(* Logix 5000 project; controller Transcat_L33ER vendor 1 type 14 code 107 rev 32.11; software revision 32.02; part 4 of 5 *)
(* tags used below, declared in another part *)
   alwaysOFF : BOOL;
   AnyAutoDeviceInterlock : BOOL;   // Any device in Auto interlocked
   AnyAutoRun : BOOL;   // Bit that in on if ANY device is placed into Auto run (to signal pre-start beed)
   AnyDeviceInterlock : BOOL;   // Any device is interlocked
   AnyManualRun : BOOL;   // Bit that in on if ANY device is placed into manual run (to signal pre-start beed)
   Auto_Run_All_Interlock : BOOL;   // Bit to interlock all devices running in Auto
   BeaconBlueLight : ALIAS FOR TC_Remote_IO:3:O.3;   // Blue Beacon Light
   BeaconGreenLight : ALIAS FOR TC_Remote_IO:3:O.2;   // Green Beacon Light
   BeaconRedLight : ALIAS FOR TC_Remote_IO:3:O.0;   // Red Beacon Light
   BeaconYellowLight : ALIAS FOR TC_Remote_IO:3:O.1;   // Yellow Beacon Light
   Beep : BOOL;   // Bit to Activte Beacon Alarm
   BeepNew : ALIAS FOR TC_Remote_IO:3:O.4;
   Device : Device[20];
   EstopActive : BOOL;   // E
   EstopFalutResetTOF : TIMER;   // Timer to hold reset bit to allow all drives to reset
   EStopReset_OS : BOOL;   // Storage bit required by the ONS instruction
   EStopResetArmed : BOOL;   // Remembers that Banner entered the waiting-for-reset state
   EStopResetPulse : BOOL;   // One-scan pulse used to clear all 14 E-stop interlocks - allows reset of estop interlocks from physical reset button on V
   FT103 : BronkhorstFlowMeter;
   FT103B : BronkhorstFlowMeter;
   FT104 : BronkhorstFlowMeter;
   FT104B : BronkhorstFlowMeter;
   FT105 : BronkhorstFlowMeter;
   FT105B : BronkhorstFlowMeter;
   GF101 : Thayer_WB_Feeder;   // Thayer 1 Tags
   GF201 : Thayer_WB_Feeder;   // Thayer 2 Tags
   GF301 : Acrison_Feeder;   // GF103 - Small Feeder 1
   GreenFlashingOff : TIMER;
   GreenFlashingOn : TIMER;
   HMI_ProcessReset : BOOL;   // Bit to clear the process hold/inteerlock when all other device interlocks are cleared
   MSG_FROM_SLC500 : INT[10];
   MX101 : Howes_Mixer;
   MX201 : Howes_Mixer;
   PT103_PV_RAW : ALIAS FOR TC_Remote_IO:1:I.Ch0Data;   // Raw (unscaled) pressure reading from PT103 - PSI * 100 (range 0 - 108 PSI)
   PT104_PV_RAW : ALIAS FOR TC_Remote_IO:1:I.Ch1Data;   // Raw (unscaled) pressure reading from PT104 - PSI * 100 (range 0 - 108 PSI)
   PT105_PV_RAW : ALIAS FOR TC_Remote_IO:1:I.Ch2Data;   // Raw (unscaled) pressure reading from PT105 - PSI * 100 (range 0 - 108 PSI)
   StartBeepTimer : TIMER;   // Timer to sound the beep alarm before starting a device
   UpperHowesSpeed : INT;
   VF101 : Acrison_Feeder;   // Medium Feeder Tags
   VF201 : Acrison_Feeder;   // Small Feeder 2 Tags
   VFD_Panel_Safety_WaitingForReset : ALIAS FOR XS26_VFD_Cabinet_Safety_Controller:I1.Data[1].5;
   YellowFlashOff : TIMER;
   YellowFlashOn : TIMER;
(* MainProgram, continued *)

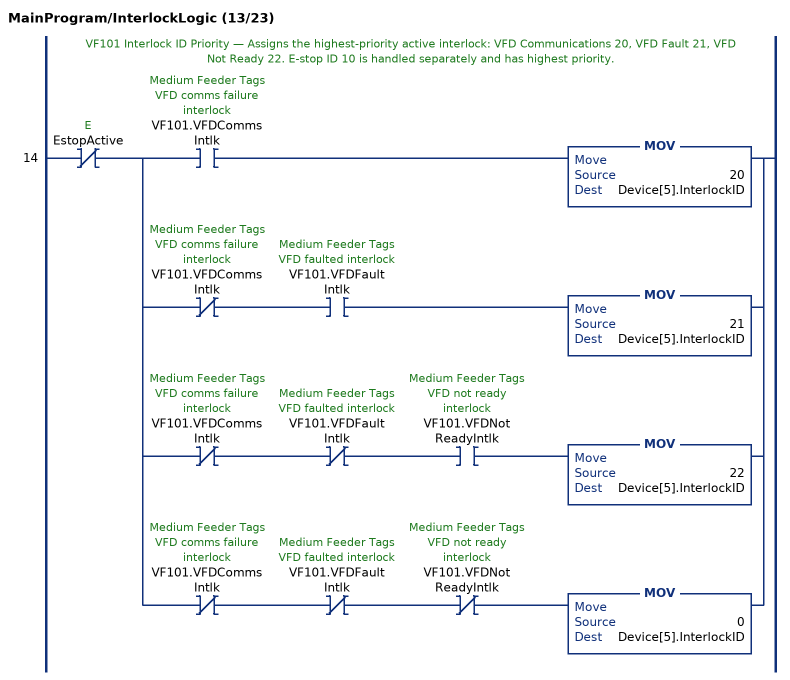
   // VF101 Interlock ID Priority — Assigns the highest-priority active interlock: VFD Communications 20, VFD Fault 21, VFD Not Ready 22. E-stop ID 10 is handled separately and has highest priority.
   14: XIO(EstopActive)[XIC(VF101.VFDCommsIntlk) MOV(20,Device[5].InterlockID) ,XIO(VF101.VFDCommsIntlk) XIC(VF101.VFDFaultIntlk) MOV(21,Device[5].InterlockID) ,XIO(VF101.VFDCommsIntlk) XIO(VF101.VFDFaultIntlk) XIC(VF101.VFDNotReadyIntlk) MOV(22,Device[5].InterlockID) ,XIO(VF101.VFDCommsIntlk) XIO(VF101.VFDFaultIntlk) XIO(VF101.VFDNotReadyIntlk) MOV(0,Device[5].InterlockID) ];
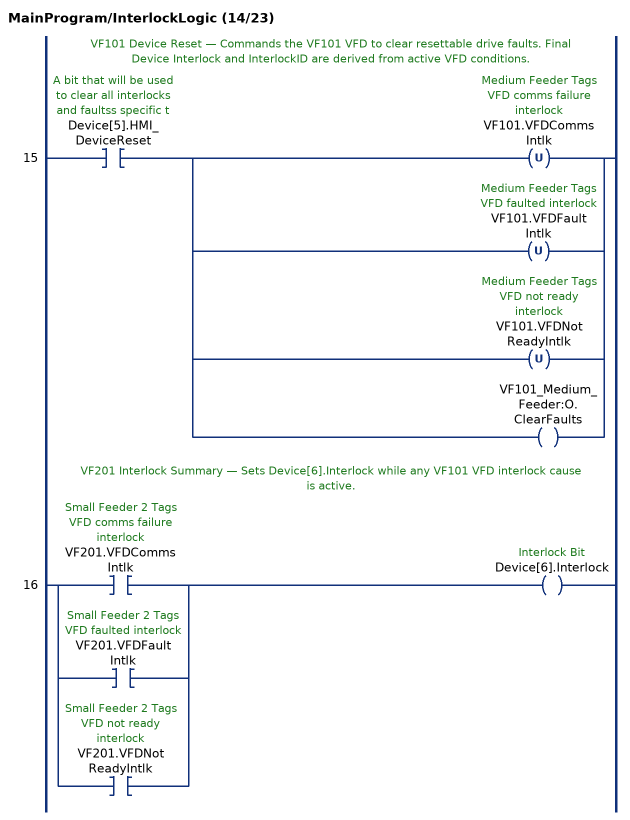
   // VF101 Device Reset — Commands the VF101 VFD to clear resettable drive faults. Final Device Interlock and InterlockID are derived from active VFD conditions.
   15: XIC(Device[5].HMI_DeviceReset)[OTU(VF101.VFDCommsIntlk) ,OTU(VF101.VFDFaultIntlk) ,OTU(VF101.VFDNotReadyIntlk) ,OTE(VF101_Medium_Feeder:O.ClearFaults) ];
   // VF201 Interlock Summary — Sets Device[6].Interlock while any VF101 VFD interlock cause is active.
   16: [XIC(VF201.VFDCommsIntlk) ,XIC(VF201.VFDFaultIntlk) ,XIC(VF201.VFDNotReadyIntlk) ]OTE(Device[6].Interlock);
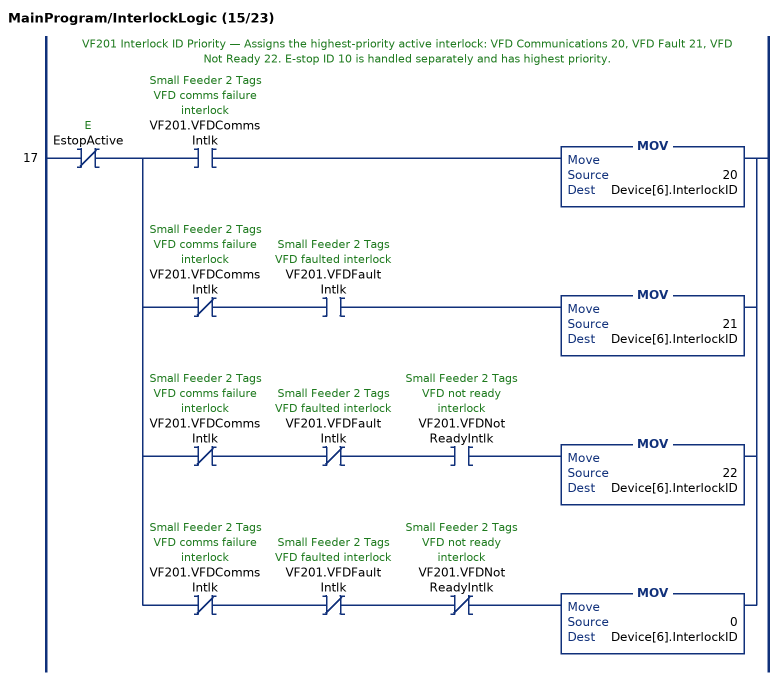
   // VF201 Interlock ID Priority — Assigns the highest-priority active interlock: VFD Communications 20, VFD Fault 21, VFD Not Ready 22. E-stop ID 10 is handled separately and has highest priority.
   17: XIO(EstopActive)[XIC(VF201.VFDCommsIntlk) MOV(20,Device[6].InterlockID) ,XIO(VF201.VFDCommsIntlk) XIC(VF201.VFDFaultIntlk) MOV(21,Device[6].InterlockID) ,XIO(VF201.VFDCommsIntlk) XIO(VF201.VFDFaultIntlk) XIC(VF201.VFDNotReadyIntlk) MOV(22,Device[6].InterlockID) ,XIO(VF201.VFDCommsIntlk) XIO(VF201.VFDFaultIntlk) XIO(VF201.VFDNotReadyIntlk) MOV(0,Device[6].InterlockID) ];
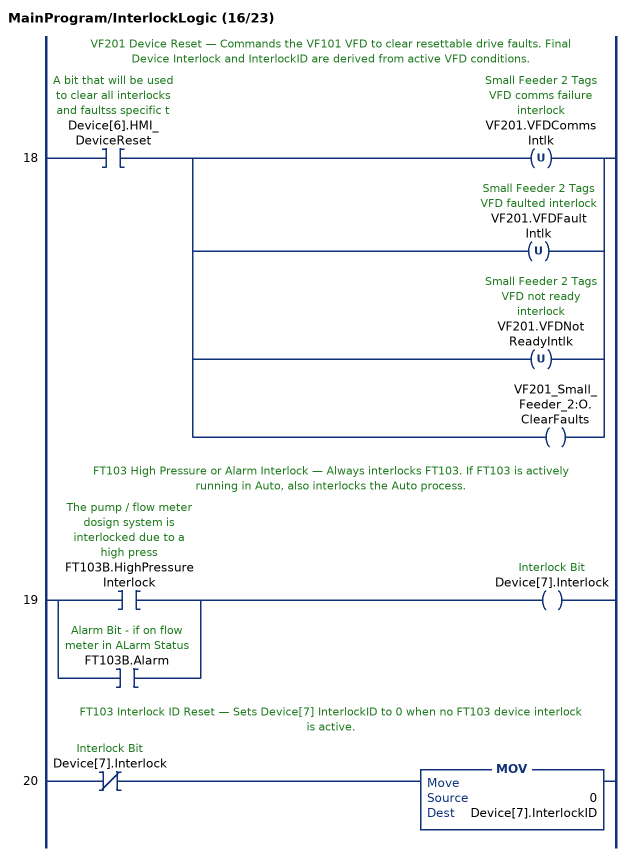
   // VF201 Device Reset — Commands the VF101 VFD to clear resettable drive faults. Final Device Interlock and InterlockID are derived from active VFD conditions.
   18: XIC(Device[6].HMI_DeviceReset)[OTU(VF201.VFDCommsIntlk) ,OTU(VF201.VFDFaultIntlk) ,OTU(VF201.VFDNotReadyIntlk) ,OTE(VF201_Small_Feeder_2:O.ClearFaults) ];
   // FT103 High Pressure or Alarm Interlock — Always interlocks FT103. If FT103 is actively running in Auto, also interlocks the Auto process.
   19: [XIC(FT103B.HighPressureInterlock) ,XIC(FT103B.Alarm) ]OTE(Device[7].Interlock);
   // FT103 Interlock ID Reset — Sets Device[7] InterlockID to 0 when no FT103 device interlock is active.
   20: XIO(Device[7].Interlock)MOV(0,Device[7].InterlockID);
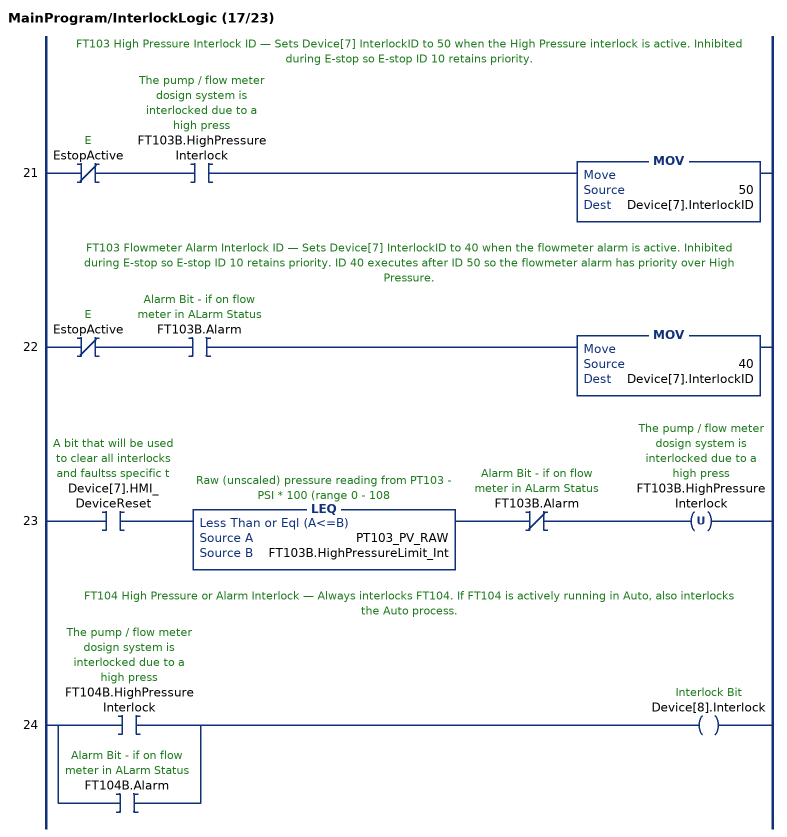
   // FT103 High Pressure Interlock ID — Sets Device[7] InterlockID to 50 when the High Pressure interlock is active. Inhibited during E-stop so E-stop ID 10 retains priority.
   21: XIO(EstopActive)XIC(FT103B.HighPressureInterlock)MOV(50,Device[7].InterlockID);
   // FT103 Flowmeter Alarm Interlock ID — Sets Device[7] InterlockID to 40 when the flowmeter alarm is active. Inhibited during E-stop so E-stop ID 10 retains priority. ID 40 executes after ID 50 so the flowmeter alarm has priority over High Pressure.
   22: XIO(EstopActive)XIC(FT103B.Alarm)MOV(40,Device[7].InterlockID);
   23: XIC(Device[7].HMI_DeviceReset)LEQ(PT103_PV_RAW,FT103B.HighPressureLimit_Int)XIO(FT103B.Alarm)OTU(FT103B.HighPressureInterlock);
   // FT104 High Pressure or Alarm Interlock — Always interlocks FT104. If FT104 is actively running in Auto, also interlocks the Auto process.
   24: [XIC(FT104B.HighPressureInterlock) ,XIC(FT104B.Alarm) ]OTE(Device[8].Interlock);
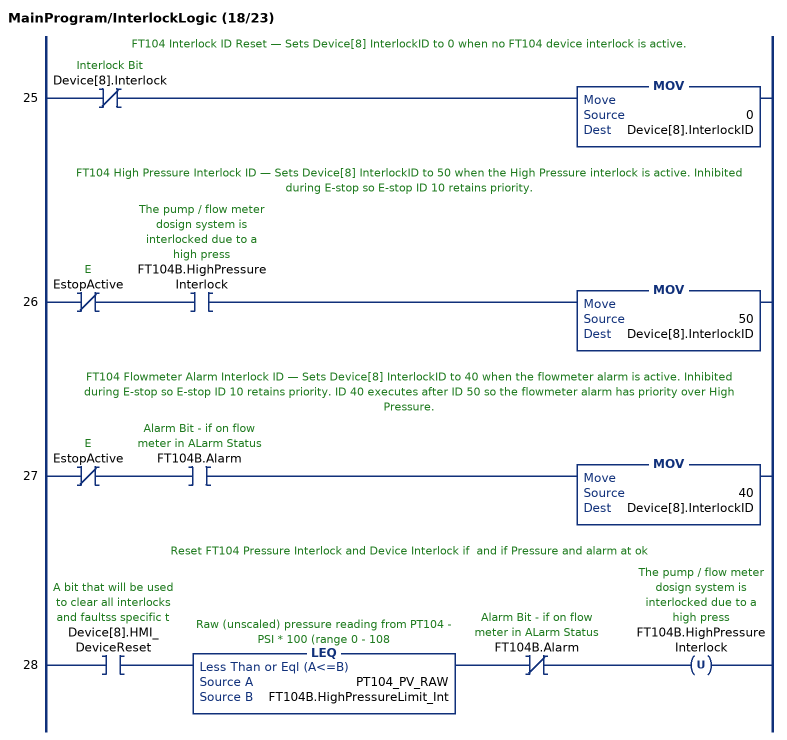
   // FT104 Interlock ID Reset — Sets Device[8] InterlockID to 0 when no FT104 device interlock is active.
   25: XIO(Device[8].Interlock)MOV(0,Device[8].InterlockID);
   // FT104 High Pressure Interlock ID — Sets Device[8] InterlockID to 50 when the High Pressure interlock is active. Inhibited during E-stop so E-stop ID 10 retains priority.
   26: XIO(EstopActive)XIC(FT104B.HighPressureInterlock)MOV(50,Device[8].InterlockID);
   // FT104 Flowmeter Alarm Interlock ID — Sets Device[8] InterlockID to 40 when the flowmeter alarm is active. Inhibited during E-stop so E-stop ID 10 retains priority. ID 40 executes after ID 50 so the flowmeter alarm has priority over High Pressure.
   27: XIO(EstopActive)XIC(FT104B.Alarm)MOV(40,Device[8].InterlockID);
   // Reset FT104 Pressure Interlock and Device Interlock if  and if Pressure and alarm at ok
   28: XIC(Device[8].HMI_DeviceReset)LEQ(PT104_PV_RAW,FT104B.HighPressureLimit_Int)XIO(FT104B.Alarm)OTU(FT104B.HighPressureInterlock);
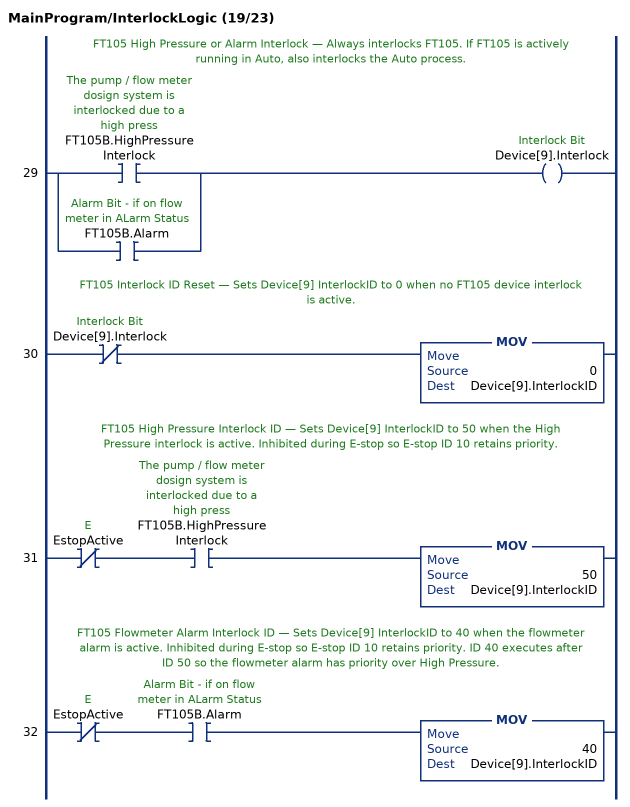
   // FT105 High Pressure or Alarm Interlock — Always interlocks FT105. If FT105 is actively running in Auto, also interlocks the Auto process.
   29: [XIC(FT105B.HighPressureInterlock) ,XIC(FT105B.Alarm) ]OTE(Device[9].Interlock);
   // FT105 Interlock ID Reset — Sets Device[9] InterlockID to 0 when no FT105 device interlock is active.
   30: XIO(Device[9].Interlock)MOV(0,Device[9].InterlockID);
   // FT105 High Pressure Interlock ID — Sets Device[9] InterlockID to 50 when the High Pressure interlock is active. Inhibited during E-stop so E-stop ID 10 retains priority.
   31: XIO(EstopActive)XIC(FT105B.HighPressureInterlock)MOV(50,Device[9].InterlockID);
   // FT105 Flowmeter Alarm Interlock ID — Sets Device[9] InterlockID to 40 when the flowmeter alarm is active. Inhibited during E-stop so E-stop ID 10 retains priority. ID 40 executes after ID 50 so the flowmeter alarm has priority over High Pressure.
   32: XIO(EstopActive)XIC(FT105B.Alarm)MOV(40,Device[9].InterlockID);
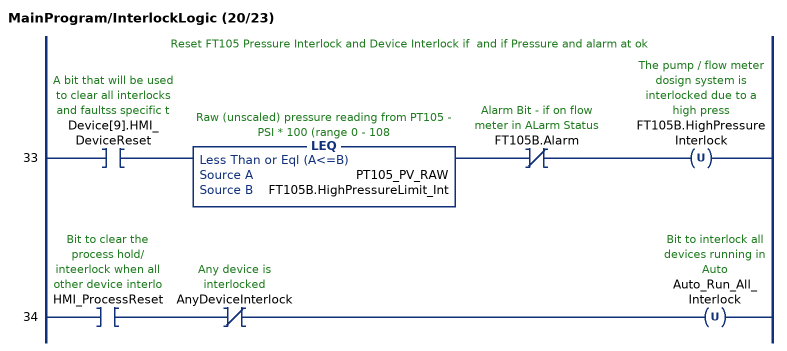
   // Reset FT105 Pressure Interlock and Device Interlock if  and if Pressure and alarm at ok
   33: XIC(Device[9].HMI_DeviceReset)LEQ(PT105_PV_RAW,FT105B.HighPressureLimit_Int)XIO(FT105B.Alarm)OTU(FT105B.HighPressureInterlock);
   34: XIC(HMI_ProcessReset)XIO(AnyDeviceInterlock)OTU(Auto_Run_All_Interlock);
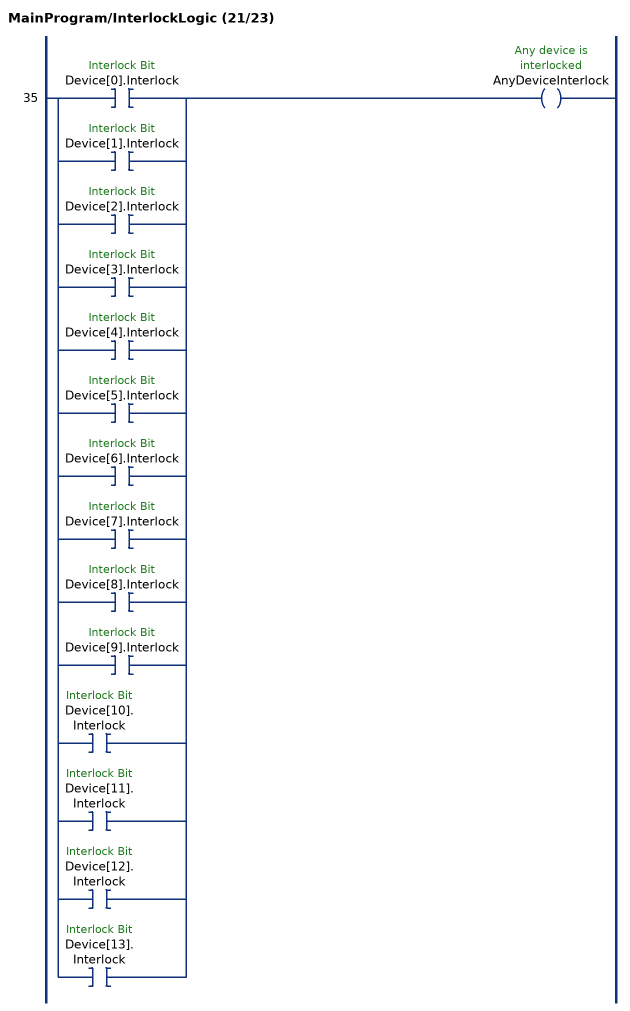
   35: [XIC(Device[0].Interlock) ,XIC(Device[1].Interlock) ,XIC(Device[2].Interlock) ,XIC(Device[3].Interlock) ,XIC(Device[4].Interlock) ,XIC(Device[5].Interlock) ,XIC(Device[6].Interlock) ,XIC(Device[7].Interlock) ,XIC(Device[8].Interlock) ,XIC(Device[9].Interlock) ,XIC(Device[10].Interlock) ,XIC(Device[11].Interlock) ,XIC(Device[12].Interlock) ,XIC(Device[13].Interlock) ]OTE(AnyDeviceInterlock);
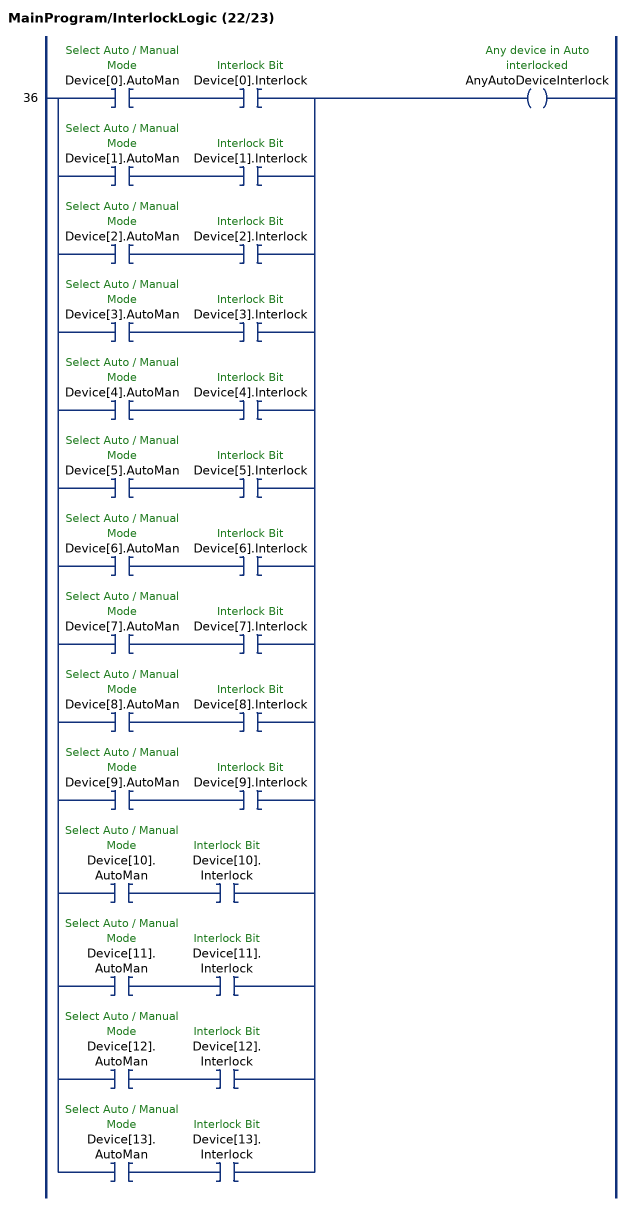
   36: [XIC(Device[0].AutoMan) XIC(Device[0].Interlock) ,XIC(Device[1].AutoMan) XIC(Device[1].Interlock) ,XIC(Device[2].AutoMan) XIC(Device[2].Interlock) ,XIC(Device[3].AutoMan) XIC(Device[3].Interlock) ,XIC(Device[4].AutoMan) XIC(Device[4].Interlock) ,XIC(Device[5].AutoMan) XIC(Device[5].Interlock) ,XIC(Device[6].AutoMan) XIC(Device[6].Interlock) ,XIC(Device[7].AutoMan) XIC(Device[7].Interlock) ,XIC(Device[8].AutoMan) XIC(Device[8].Interlock) ,XIC(Device[9].AutoMan) XIC(Device[9].Interlock) ,XIC(Device[10].AutoMan) XIC(Device[10].Interlock) ,XIC(Device[11].AutoMan) XIC(Device[11].Interlock) ,XIC(Device[12].AutoMan) XIC(Device[12].Interlock) ,XIC(Device[13].AutoMan) XIC(Device[13].Interlock) ]OTE(AnyAutoDeviceInterlock);
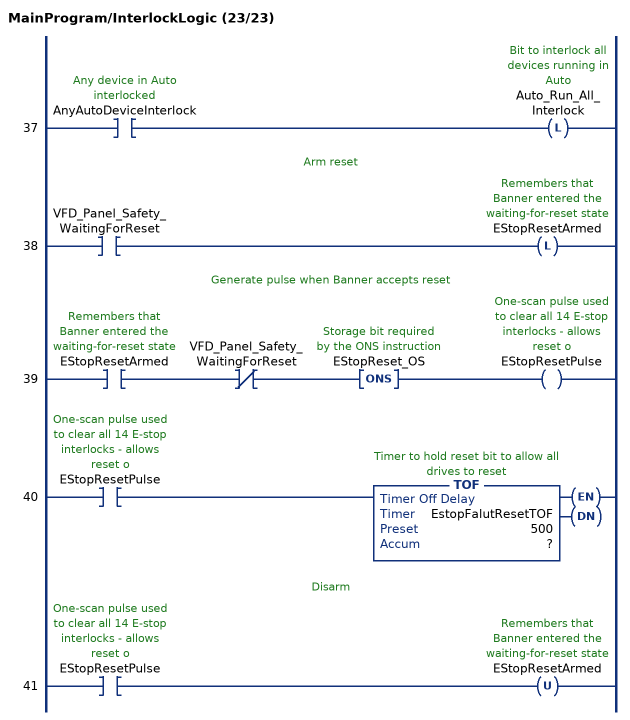
   37: XIC(AnyAutoDeviceInterlock)OTL(Auto_Run_All_Interlock);
   // Arm reset
   38: XIC(VFD_Panel_Safety_WaitingForReset)OTL(EStopResetArmed);
   // Generate pulse when Banner accepts reset
   39: XIC(EStopResetArmed)XIO(VFD_Panel_Safety_WaitingForReset)ONS(EStopReset_OS)OTE(EStopResetPulse);
   40: XIC(EStopResetPulse)TOF(EstopFalutResetTOF,?,?);
   // Disarm
   41: XIC(EStopResetPulse)OTU(EStopResetArmed);
END_ROUTINE

ROUTINE Light_Beacon   (* ladder *)
// Indicator Light Beacon
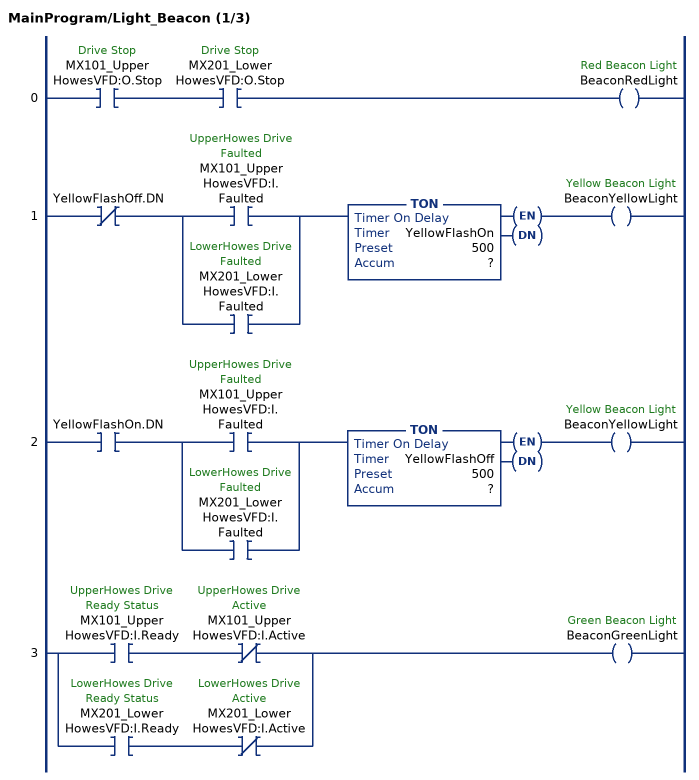
   0: XIC(MX101_UpperHowesVFD:O.Stop)XIC(MX201_LowerHowesVFD:O.Stop)OTE(BeaconRedLight);
   1: XIO(YellowFlashOff.DN)[XIC(MX101_UpperHowesVFD:I.Faulted) ,XIC(MX201_LowerHowesVFD:I.Faulted) ]TON(YellowFlashOn,?,?)OTE(BeaconYellowLight);
   2: XIC(YellowFlashOn.DN)[XIC(MX101_UpperHowesVFD:I.Faulted) ,XIC(MX201_LowerHowesVFD:I.Faulted) ]TON(YellowFlashOff,?,?)OTE(BeaconYellowLight);
   3: [XIC(MX101_UpperHowesVFD:I.Ready) XIO(MX101_UpperHowesVFD:I.Active) ,XIC(MX201_LowerHowesVFD:I.Ready) XIO(MX201_LowerHowesVFD:I.Active) ]OTE(BeaconGreenLight);
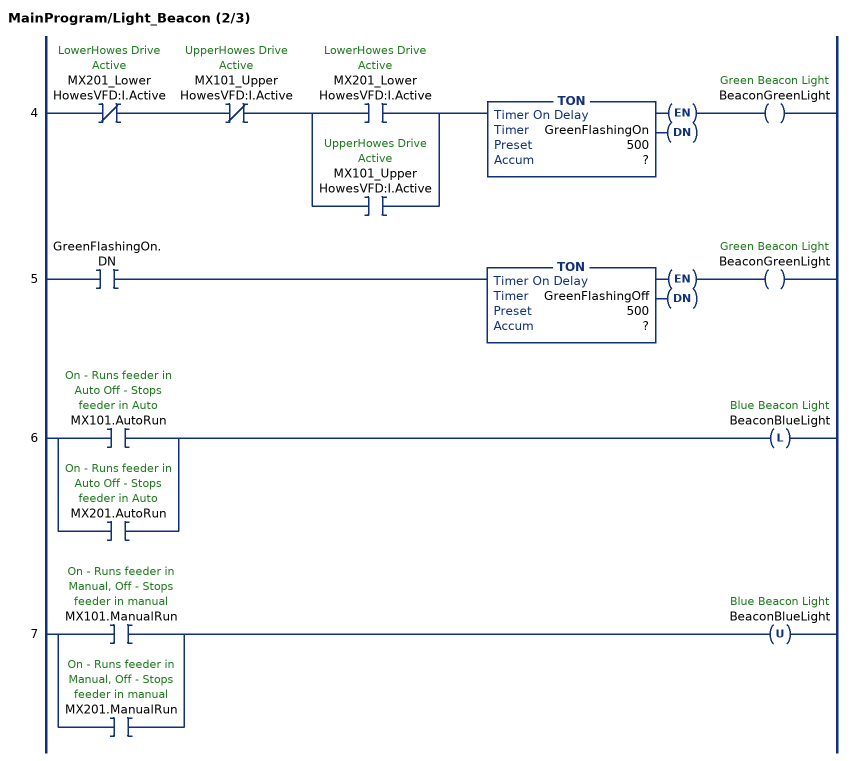
   4: XIO(MX201_LowerHowesVFD:I.Active)XIO(MX101_UpperHowesVFD:I.Active)[XIC(MX201_LowerHowesVFD:I.Active) ,XIC(MX101_UpperHowesVFD:I.Active) ]TON(GreenFlashingOn,?,?)OTE(BeaconGreenLight);
   5: XIC(GreenFlashingOn.DN)TON(GreenFlashingOff,?,?)OTE(BeaconGreenLight);
   6: [XIC(MX101.AutoRun) ,XIC(MX201.AutoRun) ]OTL(BeaconBlueLight);
   7: [XIC(MX101.ManualRun) ,XIC(MX201.ManualRun) ]OTU(BeaconBlueLight);
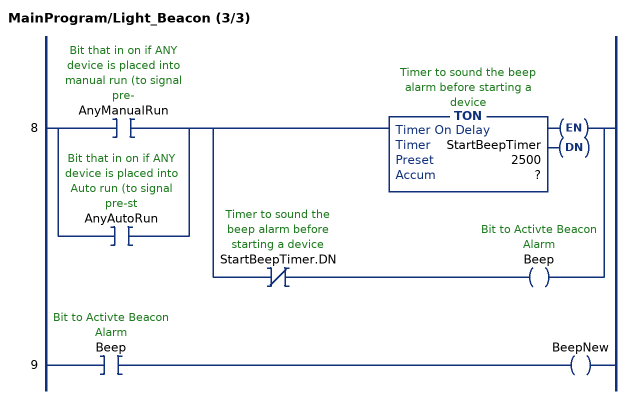
   8: [XIC(AnyManualRun) ,XIC(AnyAutoRun) ][TON(StartBeepTimer,?,?) ,XIO(StartBeepTimer.DN) OTE(Beep) ];
   9: XIC(Beep)OTE(BeepNew);
END_ROUTINE

ROUTINE MainRoutine   (* ladder *)
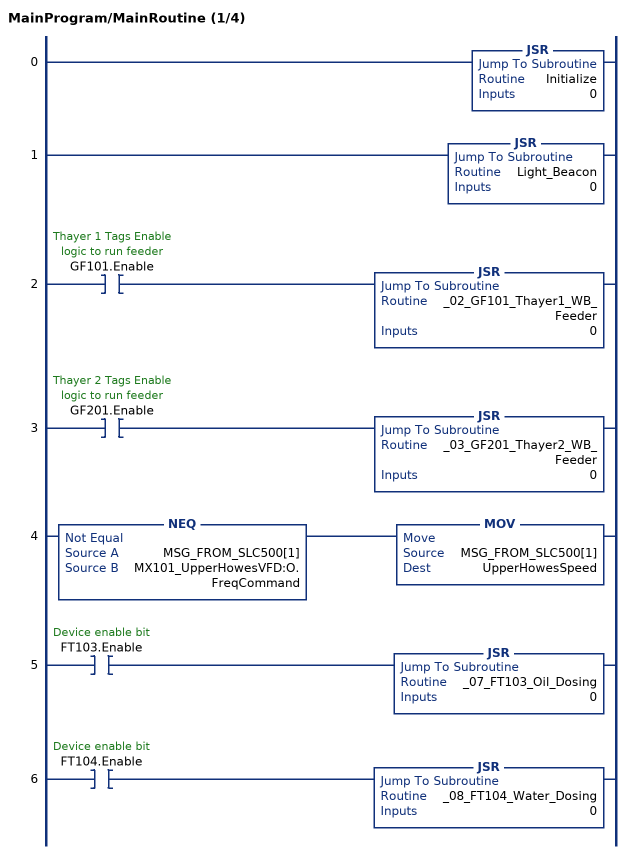
   0: JSR(Initialize,0);
   1: JSR(Light_Beacon,0);
   2: XIC(GF101.Enable)JSR(_02_GF101_Thayer1_WB_Feeder,0);
   3: XIC(GF201.Enable)JSR(_03_GF201_Thayer2_WB_Feeder,0);
   4: NEQ(MSG_FROM_SLC500[1],MX101_UpperHowesVFD:O.FreqCommand)MOV(MSG_FROM_SLC500[1],UpperHowesSpeed);
   5: XIC(FT103.Enable)JSR(_07_FT103_Oil_Dosing,0);
   6: XIC(FT104.Enable)JSR(_08_FT104_Water_Dosing,0);
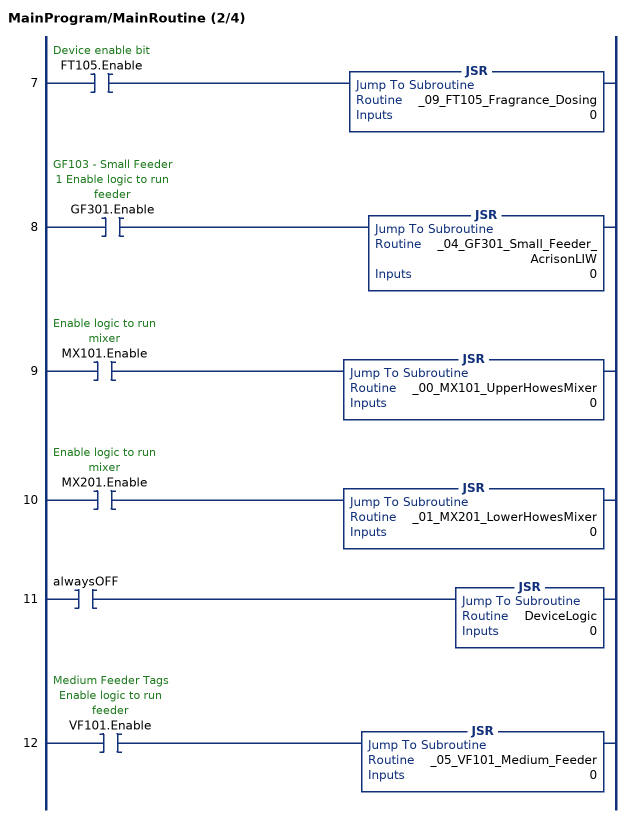
   7: XIC(FT105.Enable)JSR(_09_FT105_Fragrance_Dosing,0);
   8: XIC(GF301.Enable)JSR(_04_GF301_Small_Feeder_AcrisonLIW,0);
   9: XIC(MX101.Enable)JSR(_00_MX101_UpperHowesMixer,0);
   10: XIC(MX201.Enable)JSR(_01_MX201_LowerHowesMixer,0);
   11: XIC(alwaysOFF)JSR(DeviceLogic,0);
   12: XIC(VF101.Enable)JSR(_05_VF101_Medium_Feeder,0);
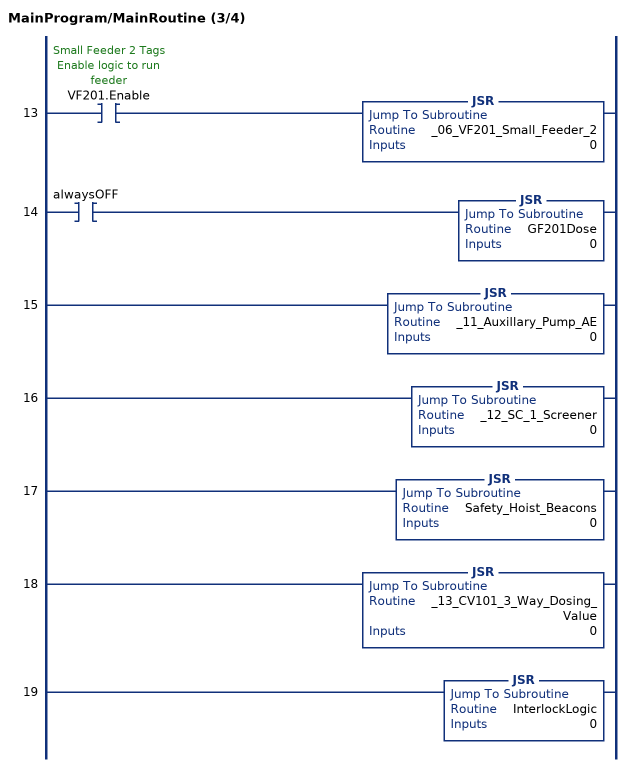
   13: XIC(VF201.Enable)JSR(_06_VF201_Small_Feeder_2,0);
   14: XIC(alwaysOFF)JSR(GF201Dose,0);
   15: JSR(_11_Auxillary_Pump_AE,0);
   16: JSR(_12_SC_1_Screener,0);
   17: JSR(Safety_Hoist_Beacons,0);
   18: JSR(_13_CV101_3_Way_Dosing_Value,0);
   19: JSR(InterlockLogic,0);
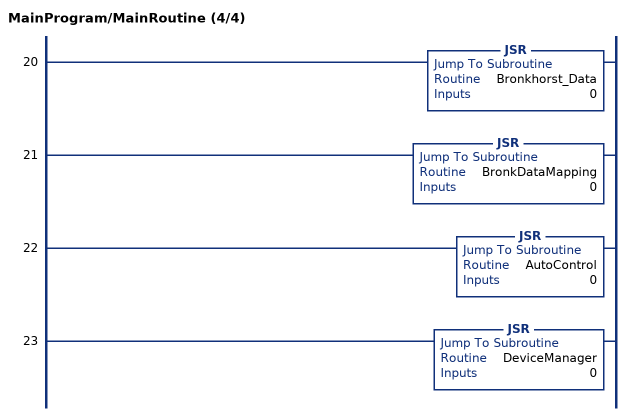
   20: JSR(Bronkhorst_Data,0);
   21: JSR(BronkDataMapping,0);
   22: JSR(AutoControl,0);
   23: JSR(DeviceManager,0);
END_ROUTINE
